PROGRAM P_SheetAlignTable
VAR
	(*Initialization*)
	bSAT_OK		: BOOL;
	bError		: BOOL;
	bStart		: BOOL;
	bStop		: BOOL;
	(*Process*)
	bBlowerEnable 	: BOOL;
	bBlowerOn		: BOOL;
	bBlowerOff		: BOOL;
	bOverride		: BOOL;
	//-----------------------------------------(*Case*)-----------------------------------------------------
	//iSATcase : INT;
	(* Reference for Sheet Align State
(
	State_Init 					,
	State_AutoStart         	,
	State_AutoStop          	,
	State_AutoBlowerOn			,
	State_AutoBackToInit        ,
	State_Override				,
	State_Error					,
);
	*)	
END_VAR
VAR_INPUT
	bStartCommand : BOOL;
	bSheetDetect	:BOOL;
END_VAR
VAR_OUTPUT
	iSATcase : INT;
	nSheetAmount	: INT;
END_VAR

bSAT_OK:=bSAT_OK;
CASE iSATcase OF

SheetAlignState.State_Init :
	bSAT_OK:=FALSE;
	IF bSAT_OK AND bStartCommand AND 
	   (NOT bError) THEN
		iSATcase:=SheetAlignState.State_AutoStart;
		bSAT_OK :=TRUE;
	ELSE
		iSATcase := SheetAlignState.State_Init;
	END_IF
	
SheetAlignState.State_AutoStart :
	(*Business Logic here*)
	iSATcase :=SheetAlignState.State_AutoBlowerOn;
	//bSAT_OK :=TRUE;

SheetAlignState.State_AutoStop :
	iSATcase :=SheetAlignState.State_Error;

SheetAlignState.State_AutoBlowerOn :
	IF bError THEN
		iSATcase :=	SheetAlignState.State_Error;
		bSAT_OK:=FALSE;
	END_IF
	IF bStop THEN
		iSATcase := SheetAlignState.State_AutoBackToInit;
	END_IF
	IF bSheetDetect THEN
		nSheetAmount:=nSheetAmount+1;
	ELSE
		nSheetAmount := nSheetAmount;
	END_IF
	
SheetAlignState.State_AutoBackToInit :
	iSATcase := SheetAlignState.State_Init;
	
SheetAlignState.State_Override :
	IF bBlowerEnable THEN
		bBlowerOn:=bBlowerOn;
		bBlowerOff:=FALSE;
	END_IF
	IF NOT bBlowerEnable THEN
		bBlowerOff:=TRUE;
	END_IF
	
SheetAlignState.State_Error :
	IF NOT bError THEN
		iSATcase := SheetAlignState.State_Error;
	END_IF
	bSAT_OK:=FALSE;
END_CASE

IF bOverride THEN
	iSATcase:= SheetAlignState.State_Override;
	bSAT_OK:=TRUE;
END_IF
IF NOT bOverride THEN
	iSATcase := iSATcase;
END_IF

END_PROGRAM

(* stored: Version 1.1.0.1, ProductVersion 3.1.4024.12
   POU P_SheetAlignTable: Id {2894f9a6-2f38-4cc2-a036-564351822d6b}, SpecialFunc None *)
